# EPICS autosave request: stdApp/Db/pvHistory.req
$(P)history$(N)_StopScan.VAL
$(P)history$(N)_Interval.B
$(P)history$(N).VALB
$(P)history$(N).VALC
$(P)history$(N).VALD
$(P)history$(N).VALE
$(P)history$(N).VALF
$(P)history$(N)_PV1_curr.INP
$(P)history$(N)_PV2_curr.INP
$(P)history$(N)_PV3_curr.INP
